FUNCTION_BLOCK FB_Trigger
VAR_INPUT
	CLK: BOOL;
END_VAR
VAR_OUTPUT
	Q: BOOL;
END_VAR
VAR
	CLK_old: BOOL;
END_VAR

IF CLK <> CLK_old AND CLK = TRUE THEN
	Q := TRUE;
ELSE
	Q := FALSE;
END_IF

CLK_old := CLK;

END_FUNCTION_BLOCK

(* stored: Version 1.1.0.1, ProductVersion 3.1.4024.12
   POU FB_Trigger: Id {bf837f36-5635-44bf-9919-774fffaad5ec}, SpecialFunc None *)
